PROGRAM HMI
VAR
	StartButtonColor:BOOL;
	SwitchOnButtonColor:BOOL;
	StopButtonColor:BOOL;
	LogoRotation:INT;
	ManualLogoRotation:INT;
	EnableManualButton:BOOL;
	
	//Timers color
	TimerColdCutColor:BOOL;
	TimerGripperPostionColor:BOOL;	
	TimerHotWeldColor:BOOL;
	TimerHeaterOnColor:BOOL;	
	StateMotorOnColor:BOOL;		
	TimerGripperopenColor:BOOL;
	TimerGripperRetractColor:BOOL;
	
	//Estop Dialog
	bOpen 						: BOOL;
	fbOpenTrigger 				: R_TRIG;
	bClose 						: BOOL;
	fbCloseTrigger 				: R_TRIG;
	EstopDialogBackgroundColor	: BOOL;
	timerDialogsBackground		:TON;
	
	TC_Restart:TC_Restart;
	
	
	//Scaling 
	onOffScaling : INT := 1000;
	WinderScaling : INT := 1000;
	IOScaling : INT := 1000;
	OutputScaling : INT := 1000;	
	SettingsScaling : INT := 1000;	
	EstopScalling	: INT := 1000;
	
	//INIT
	init:BOOL;
	timerInit:TON;
END_VAR


ACT_init();

IF init THEN
	ACT_Timers();
	IF gMachineCtrl.Simulation = FALSE THEN
		ACT_Dialogs();
	END_IF	
	
	IF gMachineCtrl.Cmd.SwitchOn THEN
		SwitchOnButtonColor := gMachineCtrl.Cmd.SwitchOn ;
	END_IF	
	
	IF gMachineCtrl.Cmd.EmStop THEN
		SwitchOnButtonColor := FALSE ;
	END_IF	
	
	IF FB_Machine_Ctrl.StepNo = 20 THEN
		LogoRotation:= (LogoRotation+5) MOD 360;
	ELSE
		//LogoRotation:=0;
	END_IF
	
	
	IF gMachineCtrl.Cmd.Manual THEN
		ManualLogoRotation:= (ManualLogoRotation+5) MOD 360;
	ELSE
		//LogoRotation:=0;
	END_IF
	
	//EnableManual Button
	IF FB_Machine_Ctrl.StepNo = 10 THEN
		EnableManualButton:=FALSE;
	ELSE
		EnableManualButton:=TRUE;
	END_IF

END_IF

TC_Restart();

ACTION ACT_Dialogs:
bOpen:= (gMachineCtrl.IO.In.E_StopPressed=TRUE);
bClose:= (gMachineCtrl.IO.In.E_StopPressed=FALSE);
//Dialog_1
//Open
fbOpenTrigger(CLK := bOpen);
IF fbOpenTrigger.Q THEN
	OpenDialog('Dialog_Estop',300,200);
END_IF
//Close
fbCloseTrigger(CLK := bClose);
IF fbCloseTrigger.Q THEN
	CloseDialog('Dialog_Estop');
END_IF

timerDialogsBackground(IN:=NOT(timerDialogsBackground.Q),PT:=T#2S);
EstopDialogBackgroundColor:= timerDialogsBackground.ET>T#1S;
END_ACTION

ACTION ACT_init:
timerInit(IN:=TRUE,PT:=T#30S);
init:=timerInit.Q;
END_ACTION

ACTION ACT_Timers:


IF FB_Machine_Run.StepNo = MACHINE_GRIPPER_END_POSITION 
OR FB_Machine_Run.StepNo = MACHINE_GRIPPER_START_POSITION THEN
	TimerGripperPostionColor:=TRUE;
ELSE
	TimerGripperPostionColor:=FALSE;
END_IF


IF FB_Machine_Run.StepNo = MACHINE_COLD_CUT_VALVE_OPEN THEN
	TimerColdCutColor:=TRUE;
ELSE
	TimerColdCutColor:=FALSE;
END_IF

IF FB_Machine_Run.StepNo = MACHINE_WELD_VALVE_OPEN
OR FB_Machine_Run.StepNo = MACHINE_VALVE_CLOSE THEN
	TimerHotWeldColor:=TRUE;
ELSE
	TimerHotWeldColor:=FALSE;
END_IF

IF FB_Machine_Run.FB_HeaterProtection.Busy
OR FB_Machine_Run.StepNo = MACHINE_HEATER_OFF THEN
	TimerHeaterOnColor:=TRUE;
ELSE
	TimerHeaterOnColor:=FALSE;
END_IF

IF FB_Machine_Run.StepNo = MACHINE_GRIPPER_OPEN
OR FB_Machine_Run.StepNo = MACHINE_GRIPPER_CLOSE THEN
	TimerGripperopenColor:=TRUE;
ELSE
	TimerGripperopenColor:=FALSE;
END_IF

IF FB_Machine_Run.StepNo = MACHINE_OUT_GRIPPER_END_POSITION OR FB_Machine_Run.StepNo = MACHINE_OUT_GRIPPER_START_POSITION THEN
	StateMotorOnColor:=TRUE;
ELSE
	StateMotorOnColor:=FALSE;
END_IF

IF FB_Machine_Run.StepNo = MACHINE_GRIPPER_RETRACT
OR FB_Machine_Run.StepNo = MACHINE_GRIPPER_EXCTRACT THEN
	TimerGripperRetractColor:=TRUE;
ELSE
	TimerGripperRetractColor:=FALSE;
END_IF
END_ACTION

END_PROGRAM

(* stored: Version 1.1.0.1, ProductVersion 3.1.4024.3
   POU HMI: Id {55836121-589d-4766-b191-c8681c6bfc5d}, SpecialFunc None
   Action ACT_Dialogs: Id {494fad89-e0ef-4d56-a0db-15a871147a1a}
   Action ACT_init: Id {6df27257-b097-423d-833f-e4b61fa64bed}
   Action ACT_Timers: Id {82e87a87-292b-4e30-a3e8-d3ae9cf93ce1} *)
